TYPE ST_P_COMPLETE_ASSY :
STRUCT
END_STRUCT
END_TYPE

(* stored: Version 1.1.0.1, ProductVersion 3.1.4024.10
   DUT ST_P_COMPLETE_ASSY: Id {3a9bee3a-15f3-4588-ad01-4865bd26560c} *)
